Fanuc KAREL source: kt00515.KL

-- PROVISIONAL review KL for V1013-1; original PC SHA256 5008643faeb6dc95e014d7af1780fdfe72d799104cba4c3a4ff99d89a0d05792
-- Incomplete behavior may be omitted. Consult companion uncertainty JSON. Do not deploy.
PROGRAM KT00515
%NOLOCKGROUP
-- UNRESOLVED_DECL P1 type=000106
-- UNRESOLVED_DECL P2 type=000101
-- UNRESOLVED_DECL OUT type=000102
BEGIN
  -- UNRESOLVED_PC offsets 5-20; opcodes 2E,22,32,35
  -- UNRESOLVED_PC offsets 25-59; opcodes 49,7E,49,60,7E,4A
  -- UNRESOLVED_PC offsets 64-68; opcodes 7F
END KT00515
